TYPE E_GPInputMode :
(
	Disabled,
	Analog,
	Digital,
	Limits
);
END_TYPE

(* stored: Version 1.1.0.1, ProductVersion 3.1.4022.10
   DUT E_GPInputMode: Id {08b2e105-41c1-4b80-8935-4b439debf6bd} *)
